Fanuc KAREL source: ko00065.KL

PROGRAM KO00065
%STACKSIZE=65535
%PRIORITY=65535
%NOLOCKGROUP
VAR
P1 : XYZWPREXT
P2 : POSITION
F : BOOLEAN
OUT : POSITION
BEGIN
F=TRUE
-- UNSAFE_SOURCE_IR line 11: CALL_RESULT MIRROR(P1, P2, F)
END KO00065
